TYPE ST_SchrauberAblauf_AchsStruc :
STRUCT
	(*========================================================================================================================*)
	(* === Achsstruktur INOUT === *)
	(*========================================================================================================================*)
	NC_Axis_OUT_bSteuerwortBit1			:BOOL;
	NC_Axis_OUT_bSteuerwortBit2			:BOOL;
	
	NC_Axis_OUT_bIstwertSetzen			:BOOL;
	NC_Axis_OUT_bAchsePosStarten		:BOOL;
	NC_Axis_OUT_bAchsePosStoppen		:BOOL;
	NC_Axis_OUT_nPosIstwertSetzen		:LREAL;
	NC_Axis_OUT_nPTPVelo				:LREAL;
	NC_Axis_OUT_PTPBuffMode				:MC_BufferMode;
	
	NC_Axis_IN_bDCStatuswort13			:BOOL;
	NC_Axis_IN_bStatuswortBit0			:BOOL;
	NC_Axis_IN_bIstWertgesetzt			:BOOL;
	NC_Axis_IN_bPTPPosiFreig			:BOOL;
	NC_Axis_IN_bNcFehler				:BOOL;
	NC_Axis_IN_nActPos					:LREAL;
	NC_Axis_IN_nActVelo					:LREAL;
	NC_Axis_IN_nParamEilgeschw			:LREAL;
	NC_Axis_IN_nActTorque				:INT;
	
	NC_Axis_IN_bFaehrtPos				:BOOL;
	NC_Axis_IN_bInPos					:BOOL;
	NC_Axis_IN_bInStillstand			:BOOL;
	
END_STRUCT
END_TYPE

(* stored: Version 1.1.0.1, ProductVersion 3.1.4024.15
   DUT ST_SchrauberAblauf_AchsStruc: Id {379bbe5d-8a1a-4b00-a37d-b5a7f8c7ac25} *)
